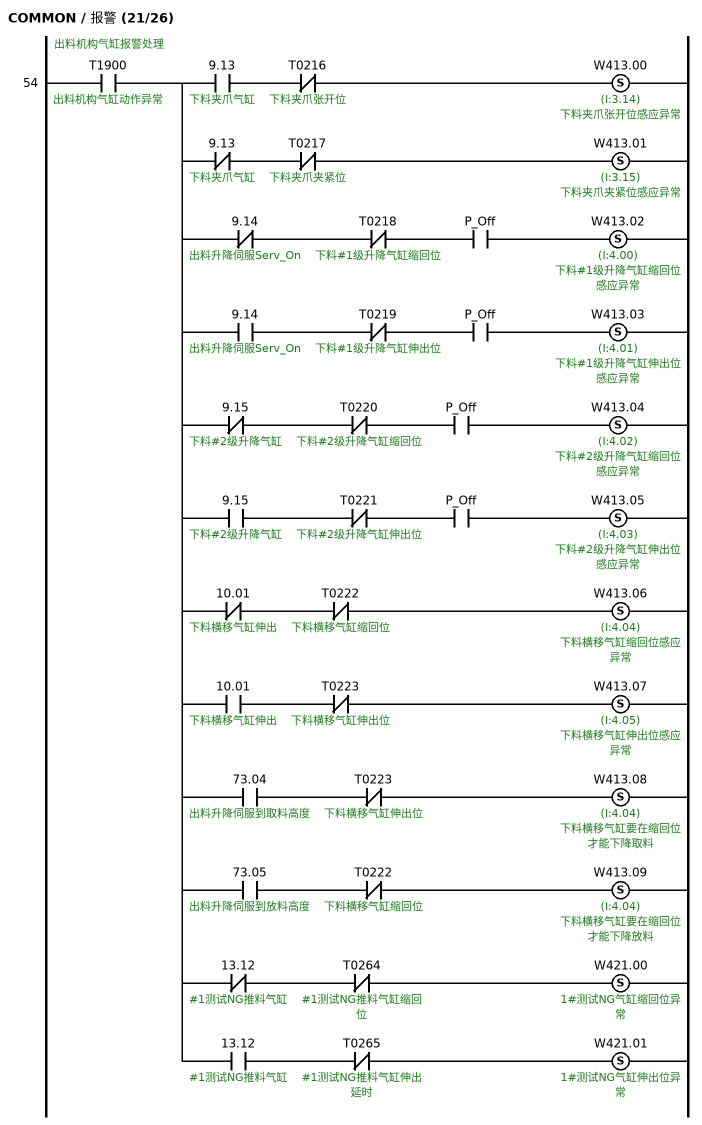
; [picture p456: COMMON / 报警, rungs 54-54]
; rung 54: 出料机构气缸报警处理
LD T1900  ; 出料机构气缸动作异常
OUT TR0
AND 9.13  ; 下料夹爪气缸
ANDNOT T0216  ; 下料夹爪张开位
SET W413.00  ; (I:3.14) 下料夹爪张开位感应异常
LD TR0
ANDNOT 9.13  ; 下料夹爪气缸
ANDNOT T0217  ; 下料夹爪夹紧位
SET W413.01  ; (I:3.15) 下料夹爪夹紧位感应异常
LD TR0
ANDNOT 9.14  ; 出料升降伺服Serv_On
ANDNOT T0218  ; 下料#1级升降气缸缩回位
AND P_Off
SET W413.02  ; (I:4.00) 下料#1级升降气缸缩回位感应异常
LD TR0
AND 9.14  ; 出料升降伺服Serv_On
ANDNOT T0219  ; 下料#1级升降气缸伸出位
AND P_Off
SET W413.03  ; (I:4.01) 下料#1级升降气缸伸出位感应异常
LD TR0
ANDNOT 9.15  ; 下料#2级升降气缸
ANDNOT T0220  ; 下料#2级升降气缸缩回位
AND P_Off
SET W413.04  ; (I:4.02) 下料#2级升降气缸缩回位感应异常
LD TR0
AND 9.15  ; 下料#2级升降气缸
ANDNOT T0221  ; 下料#2级升降气缸伸出位
AND P_Off
SET W413.05  ; (I:4.03) 下料#2级升降气缸伸出位感应异常
LD TR0
ANDNOT 10.01  ; 下料横移气缸伸出
ANDNOT T0222  ; 下料横移气缸缩回位
SET W413.06  ; (I:4.04) 下料横移气缸缩回位感应异常
LD TR0
AND 10.01  ; 下料横移气缸伸出
ANDNOT T0223  ; 下料横移气缸伸出位
SET W413.07  ; (I:4.05) 下料横移气缸伸出位感应异常
LD TR0
AND 73.04  ; 出料升降伺服到取料高度
ANDNOT T0223  ; 下料横移气缸伸出位
SET W413.08  ; (I:4.04) 下料横移气缸要在缩回位才能下降取料
LD TR0
AND 73.05  ; 出料升降伺服到放料高度
ANDNOT T0222  ; 下料横移气缸缩回位
SET W413.09  ; (I:4.04) 下料横移气缸要在缩回位才能下降放料
LD TR0
ANDNOT 13.12  ; #1测试NG推料气缸
ANDNOT T0264  ; #1测试NG推料气缸缩回位
SET W421.00  ; 1#测试NG气缸缩回位异常
LD TR0
AND 13.12  ; #1测试NG推料气缸
ANDNOT T0265  ; #1测试NG推料气缸伸出延时
SET W421.01  ; 1#测试NG气缸伸出位异常

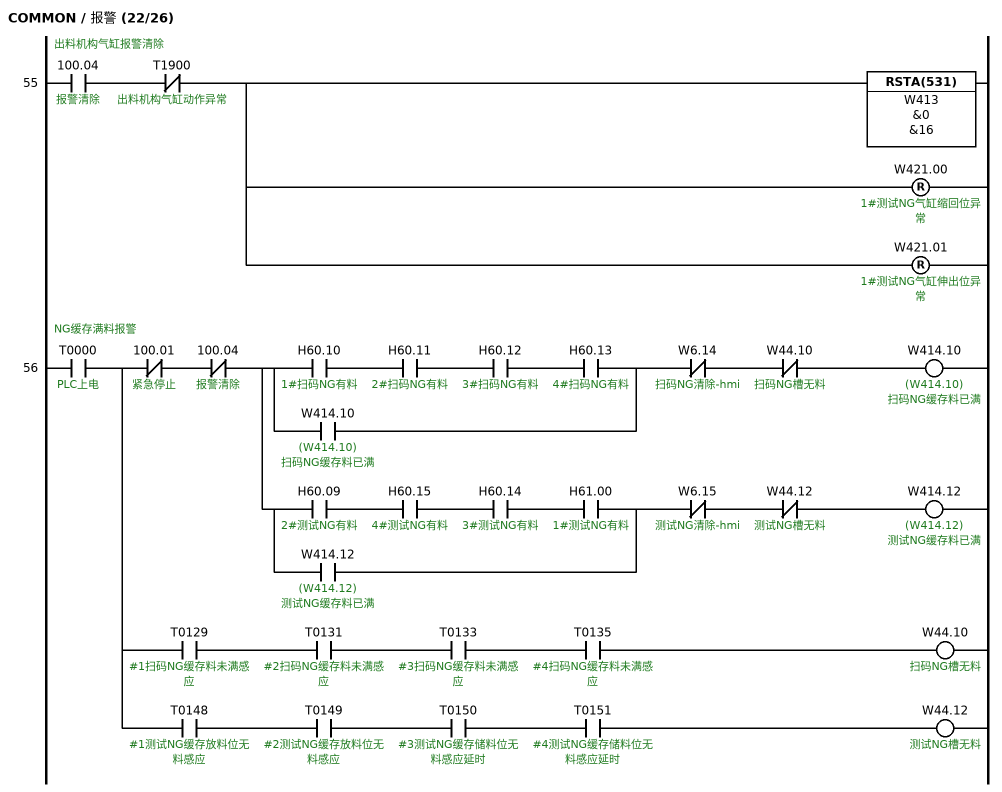
; rung 55: 出料机构气缸报警清除
LD 100.04  ; 报警清除
ANDNOT T1900  ; 出料机构气缸动作异常
RSTA(531) W413 &0 &16
RSET W421.00  ; 1#测试NG气缸缩回位异常
RSET W421.01  ; 1#测试NG气缸伸出位异常
; rung 56: NG缓存满料报警
LD T0000  ; PLC上电
OUT TR0
ANDNOT 100.01  ; 紧急停止
ANDNOT 100.04  ; 报警清除
OUT TR1
LD H60.10  ; 1#扫码NG有料
AND H60.11  ; 2#扫码NG有料
AND H60.12  ; 3#扫码NG有料
AND H60.13  ; 4#扫码NG有料
OR W414.10  ; (W414.10) 扫码NG缓存料已满
ANDLD
ANDNOT W6.14  ; 扫码NG清除-hmi
ANDNOT W44.10  ; 扫码NG槽无料
OUT W414.10  ; (W414.10) 扫码NG缓存料已满
LD TR1
LD H60.09  ; 2#测试NG有料
AND H60.15  ; 4#测试NG有料
AND H60.14  ; 3#测试NG有料
AND H61.00  ; 1#测试NG有料
OR W414.12  ; (W414.12) 测试NG缓存料已满
ANDLD
ANDNOT W6.15  ; 测试NG清除-hmi
ANDNOT W44.12  ; 测试NG槽无料
OUT W414.12  ; (W414.12) 测试NG缓存料已满
LD TR0
AND T0129  ; #1扫码NG缓存料未满感应
AND T0131  ; #2扫码NG缓存料未满感应
AND T0133  ; #3扫码NG缓存料未满感应
AND T0135  ; #4扫码NG缓存料未满感应
OUT W44.10  ; 扫码NG槽无料
LD TR0
AND T0148  ; #1测试NG缓存放料位无料感应
AND T0149  ; #2测试NG缓存放料位无料感应
AND T0150  ; #3测试NG缓存储料位无料感应延时
AND T0151  ; #4测试NG缓存储料位无料感应延时
OUT W44.12  ; 测试NG槽无料

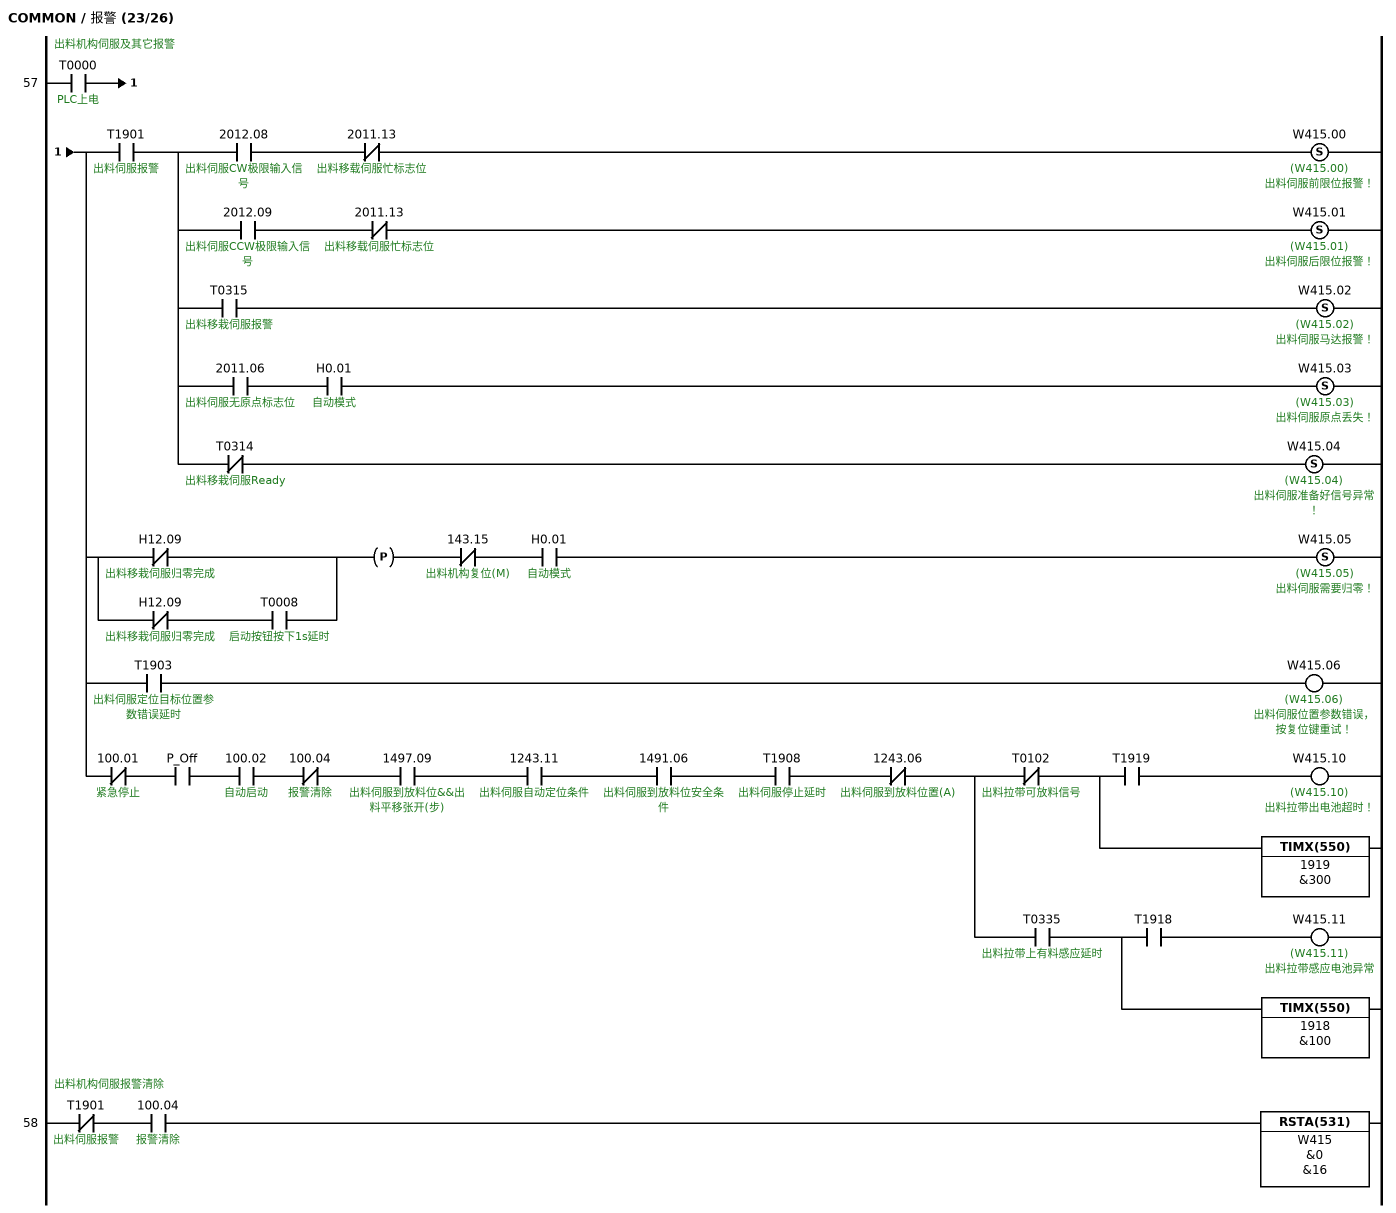
; rung 57: 出料机构伺服及其它报警
LD T0000  ; PLC上电
OUT TR0
AND T1901  ; 出料伺服报警
OUT TR1
AND 2012.08  ; 出料伺服CW极限输入信号
ANDNOT 2011.13  ; 出料移载伺服忙标志位
SET W415.00  ; (W415.00) 出料伺服前限位报警！
LD TR1
AND 2012.09  ; 出料伺服CCW极限输入信号
ANDNOT 2011.13  ; 出料移载伺服忙标志位
SET W415.01  ; (W415.01) 出料伺服后限位报警！
LD TR1
AND T0315  ; 出料移栽伺服报警
SET W415.02  ; (W415.02) 出料伺服马达报警！
LD TR1
AND 2011.06  ; 出料伺服无原点标志位
AND H0.01  ; 自动模式
SET W415.03  ; (W415.03) 出料伺服原点丢失！
LD TR1
ANDNOT T0314  ; 出料移栽伺服Ready
SET W415.04  ; (W415.04) 出料伺服准备好信号异常！
LD TR0
LDNOT H12.09  ; 出料移栽伺服归零完成
LDNOT H12.09  ; 出料移栽伺服归零完成
AND T0008  ; 启动按钮按下1s延时
ORLD
ANDLD
UP(521)
ANDNOT 143.15  ; 出料机构复位(M)
AND H0.01  ; 自动模式
SET W415.05  ; (W415.05) 出料伺服需要归零！
LD TR0
AND T1903  ; 出料伺服定位目标位置参数错误延时
OUT W415.06  ; (W415.06) 出料伺服位置参数错误，按复位键重试！
LD TR0
ANDNOT 100.01  ; 紧急停止
AND P_Off
AND 100.02  ; 自动启动
ANDNOT 100.04  ; 报警清除
AND 1497.09  ; 出料伺服到放料位&&出料平移张开(步)
AND 1243.11  ; 出料伺服自动定位条件
AND 1491.06  ; 出料伺服到放料位安全条件
AND T1908  ; 出料伺服停止延时
ANDNOT 1243.06  ; 出料伺服到放料位置(A)
OUT TR0
ANDNOT T0102  ; 出料拉带可放料信号
OUT TR1
AND T1919
OUT W415.10  ; (W415.10) 出料拉带出电池超时！
LD TR1
TIMX(550) 1919 &300
LD TR0
AND T0335  ; 出料拉带上有料感应延时
OUT TR0
AND T1918
OUT W415.11  ; (W415.11) 出料拉带感应电池异常
LD TR0
TIMX(550) 1918 &100
; rung 58: 出料机构伺服报警清除
LDNOT T1901  ; 出料伺服报警
AND 100.04  ; 报警清除
RSTA(531) W415 &0 &16

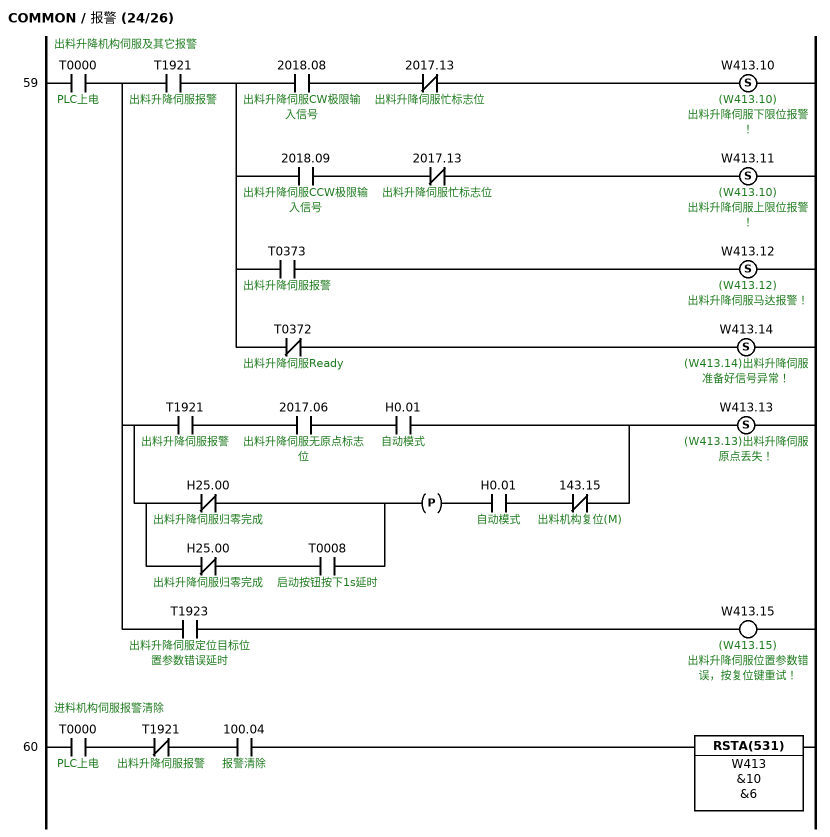
; rung 59: 出料升降机构伺服及其它报警
LD T0000  ; PLC上电
OUT TR0
AND T1921  ; 出料升降伺服报警
OUT TR1
AND 2018.08  ; 出料升降伺服CW极限输入信号
ANDNOT 2017.13  ; 出料升降伺服忙标志位
SET W413.10  ; (W413.10) 出料升降伺服下限位报警！
LD TR1
AND 2018.09  ; 出料升降伺服CCW极限输入信号
ANDNOT 2017.13  ; 出料升降伺服忙标志位
SET W413.11  ; (W413.10) 出料升降伺服上限位报警！
LD TR1
AND T0373  ; 出料升降伺服报警
SET W413.12  ; (W413.12) 出料升降伺服马达报警！
LD TR1
ANDNOT T0372  ; 出料升降伺服Ready
SET W413.14  ; (W413.14)出料升降伺服准备好信号异常！
LD TR0
LD T1921  ; 出料升降伺服报警
AND 2017.06  ; 出料升降伺服无原点标志位
AND H0.01  ; 自动模式
LDNOT H25.00  ; 出料升降伺服归零完成
LDNOT H25.00  ; 出料升降伺服归零完成
AND T0008  ; 启动按钮按下1s延时
ORLD
UP(521)
AND H0.01  ; 自动模式
ANDNOT 143.15  ; 出料机构复位(M)
ORLD
ANDLD
SET W413.13  ; (W413.13)出料升降伺服原点丢失！
LD TR0
AND T1923  ; 出料升降伺服定位目标位置参数错误延时
OUT W413.15  ; (W413.15) 出料升降伺服位置参数错误，按复位键重试！
; rung 60: 进料机构伺服报警清除
LD T0000  ; PLC上电
ANDNOT T1921  ; 出料升降伺服报警
AND 100.04  ; 报警清除
RSTA(531) W413 &10 &6

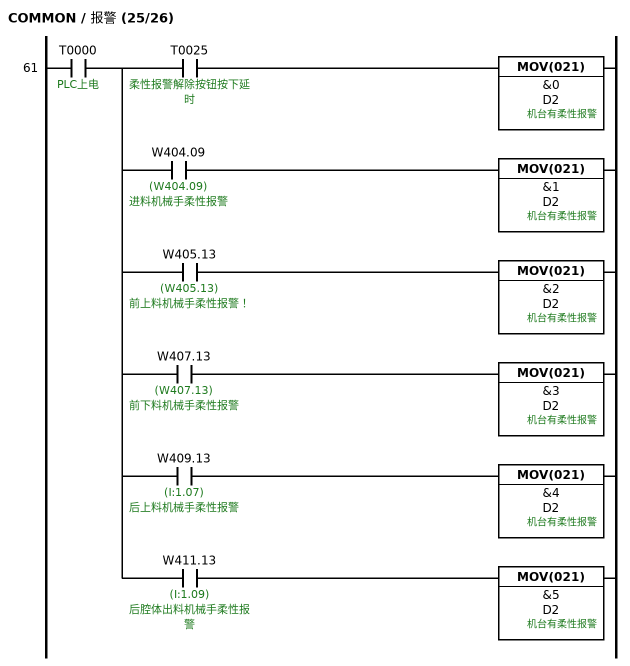
; rung 61
LD T0000  ; PLC上电
OUT TR0
AND T0025  ; 柔性报警解除按钮按下延时
MOV(021) &0 D2  ; 机台有柔性报警
LD TR0
AND W404.09  ; (W404.09) 进料机械手柔性报警
MOV(021) &1 D2  ; 机台有柔性报警
LD TR0
AND W405.13  ; (W405.13) 前上料机械手柔性报警！
MOV(021) &2 D2  ; 机台有柔性报警
LD TR0
AND W407.13  ; (W407.13) 前下料机械手柔性报警
MOV(021) &3 D2  ; 机台有柔性报警
LD TR0
AND W409.13  ; (I:1.07) 后上料机械手柔性报警
MOV(021) &4 D2  ; 机台有柔性报警
LD TR0
AND W411.13  ; (I:1.09) 后腔体出料机械手柔性报警
MOV(021) &5 D2  ; 机台有柔性报警

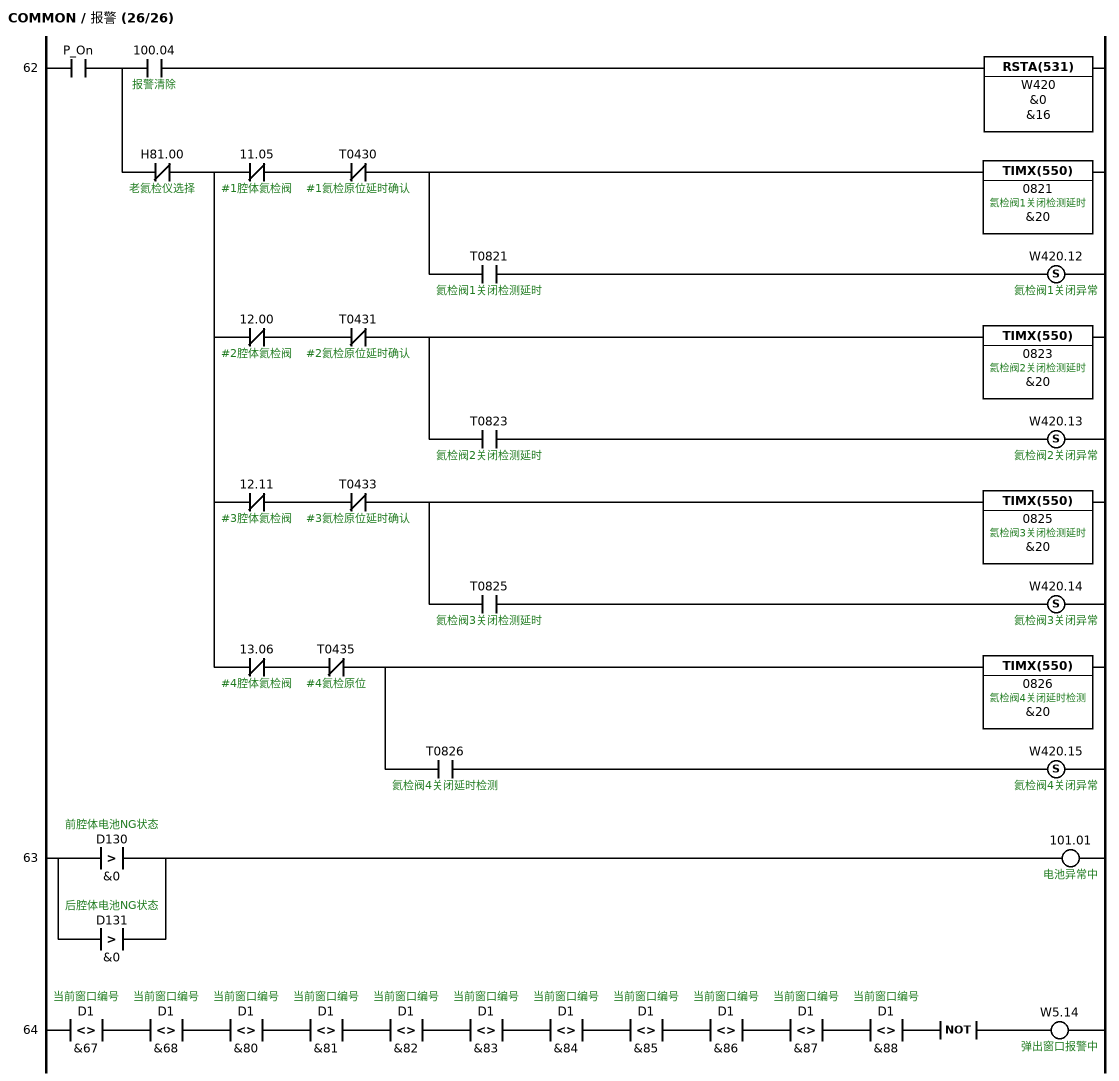
; rung 62
LD P_On
OUT TR0
AND 100.04  ; 报警清除
RSTA(531) W420 &0 &16
LD TR0
ANDNOT H81.00  ; 老氦检仪选择
OUT TR0
ANDNOT 11.05  ; #1腔体氦检阀
ANDNOT T0430  ; #1氦检原位延时确认
TIMX(550) 0821 &20  ; 氦检阀1关闭检测延时
AND T0821  ; 氦检阀1关闭检测延时
SET W420.12  ; 氦检阀1关闭异常
LD TR0
ANDNOT 12.00  ; #2腔体氦检阀
ANDNOT T0431  ; #2氦检原位延时确认
TIMX(550) 0823 &20  ; 氦检阀2关闭检测延时
AND T0823  ; 氦检阀2关闭检测延时
SET W420.13  ; 氦检阀2关闭异常
LD TR0
ANDNOT 12.11  ; #3腔体氦检阀
ANDNOT T0433  ; #3氦检原位延时确认
TIMX(550) 0825 &20  ; 氦检阀3关闭检测延时
AND T0825  ; 氦检阀3关闭检测延时
SET W420.14  ; 氦检阀3关闭异常
LD TR0
ANDNOT 13.06  ; #4腔体氦检阀
ANDNOT T0435  ; #4氦检原位
TIMX(550) 0826 &20  ; 氦检阀4关闭延时检测
AND T0826  ; 氦检阀4关闭延时检测
SET W420.15  ; 氦检阀4关闭异常
; rung 63
LD>(320) D130 &0  ; 前腔体电池NG状态
OR>(320) D131 &0  ; 后腔体电池NG状态
OUT 101.01  ; 电池异常中
; rung 64
LD<>(305) D1 &67  ; 当前窗口编号
AND<>(305) D1 &68  ; 当前窗口编号
AND<>(305) D1 &80  ; 当前窗口编号
AND<>(305) D1 &81  ; 当前窗口编号
AND<>(305) D1 &82  ; 当前窗口编号
AND<>(305) D1 &83  ; 当前窗口编号
AND<>(305) D1 &84  ; 当前窗口编号
AND<>(305) D1 &85  ; 当前窗口编号
AND<>(305) D1 &86  ; 当前窗口编号
AND<>(305) D1 &87  ; 当前窗口编号
AND<>(305) D1 &88  ; 当前窗口编号
NOT(520)
OUT W5.14  ; 弹出窗口报警中

### Section 数据传递

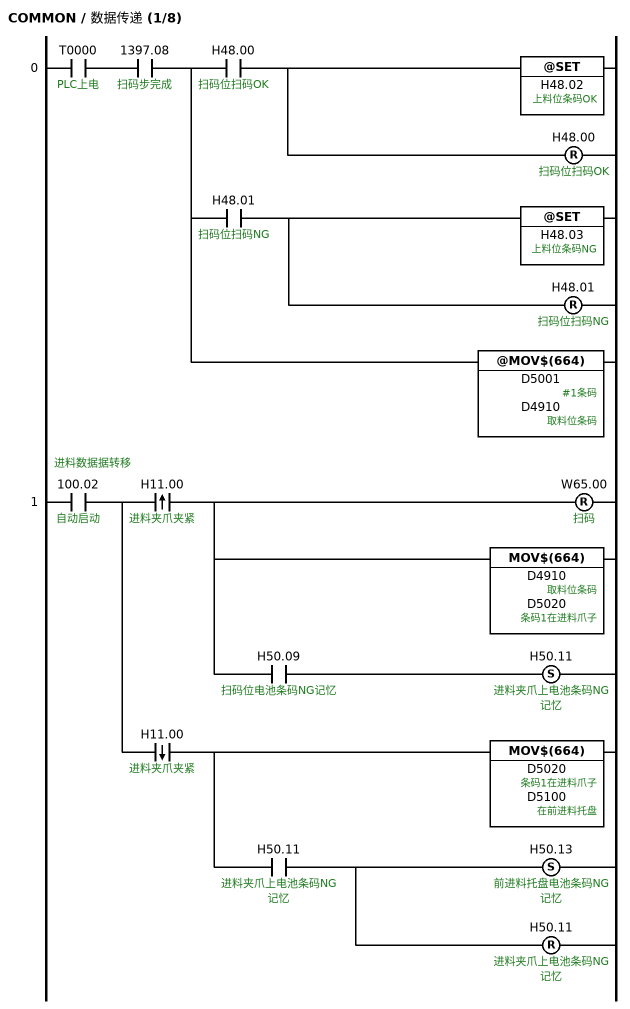
; rung 0
LD T0000  ; PLC上电
AND 1397.08  ; 扫码步完成
OUT TR0
AND H48.00  ; 扫码位扫码OK
@SET H48.02  ; 上料位条码OK
RSET H48.00  ; 扫码位扫码OK
LD TR0
AND H48.01  ; 扫码位扫码NG
@SET H48.03  ; 上料位条码NG
RSET H48.01  ; 扫码位扫码NG
LD TR0
@MOV$(664) D5001 D4910  ; #1条码, 取料位条码
; rung 1: 进料数据据转移
LD 100.02  ; 自动启动
OUT TR0
@AND H11.00  ; 进料夹爪夹紧
RSET W65.00  ; 扫码
MOV$(664) D4910 D5020  ; 取料位条码, 条码1在进料爪子
AND H50.09  ; 扫码位电池条码NG记忆
SET H50.11  ; 进料夹爪上电池条码NG记忆
LD TR0
%AND H11.00  ; 进料夹爪夹紧
MOV$(664) D5020 D5100  ; 条码1在进料爪子, 在前进料托盘
AND H50.11  ; 进料夹爪上电池条码NG记忆
SET H50.13  ; 前进料托盘电池条码NG记忆
RSET H50.11  ; 进料夹爪上电池条码NG记忆

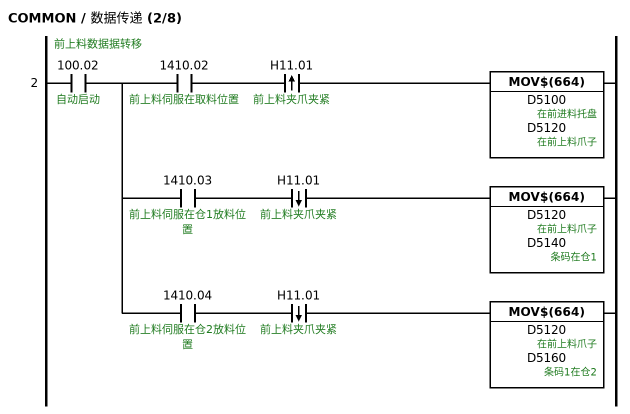
; rung 2: 前上料数据据转移
LD 100.02  ; 自动启动
OUT TR0
AND 1410.02  ; 前上料伺服在取料位置
@AND H11.01  ; 前上料夹爪夹紧
MOV$(664) D5100 D5120  ; 在前进料托盘, 在前上料爪子
LD TR0
AND 1410.03  ; 前上料伺服在仓1放料位置
%AND H11.01  ; 前上料夹爪夹紧
MOV$(664) D5120 D5140  ; 在前上料爪子, 条码在仓1
LD TR0
AND 1410.04  ; 前上料伺服在仓2放料位置
%AND H11.01  ; 前上料夹爪夹紧
MOV$(664) D5120 D5160  ; 在前上料爪子, 条码1在仓2

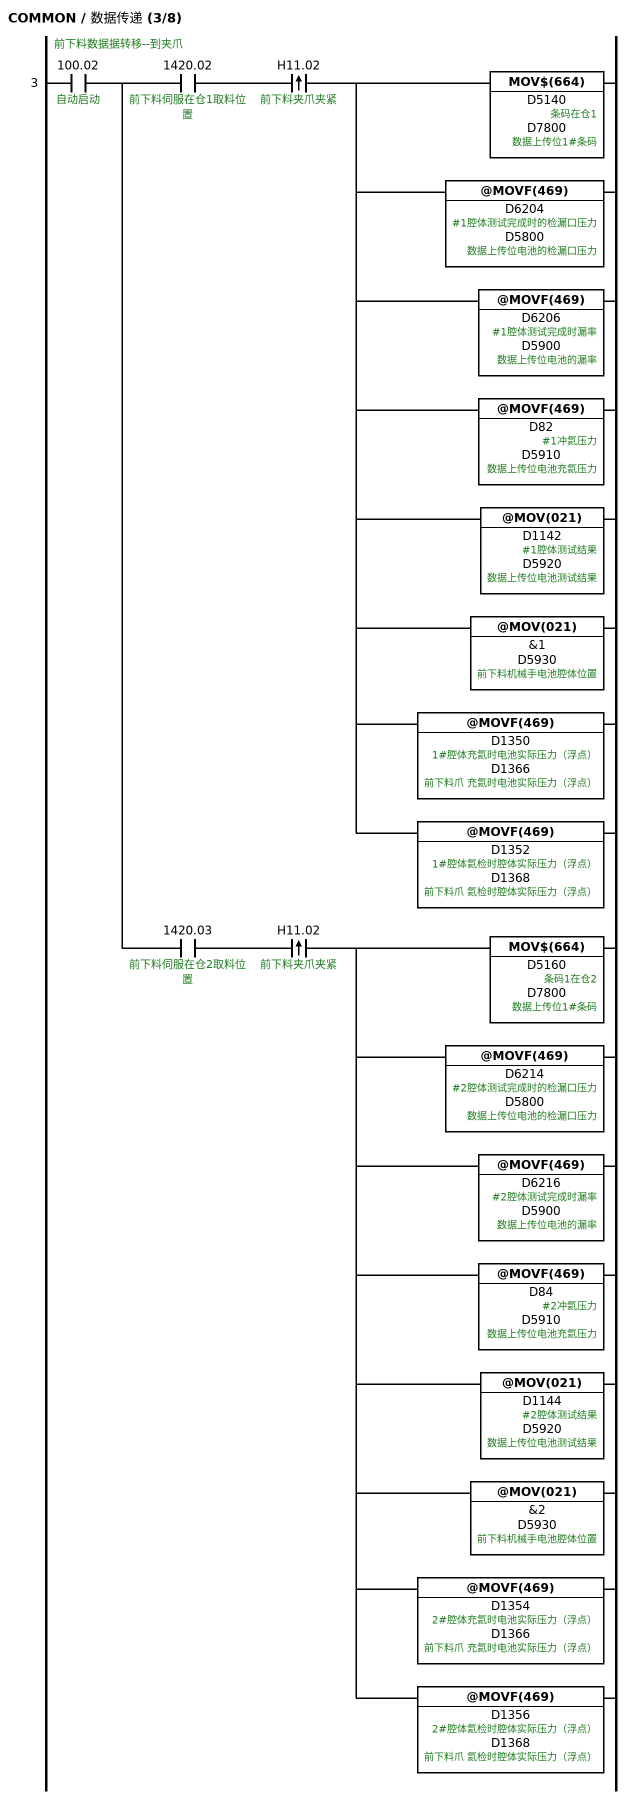
; rung 3: 前下料数据据转移--到夹爪
LD 100.02  ; 自动启动
OUT TR0
AND 1420.02  ; 前下料伺服在仓1取料位置
@AND H11.02  ; 前下料夹爪夹紧
MOV$(664) D5140 D7800  ; 条码在仓1, 数据上传位1#条码
@MOVF(469) D6204 D5800  ; #1腔体测试完成时的检漏口压力, 数据上传位电池的检漏口压力
@MOVF(469) D6206 D5900  ; #1腔体测试完成时漏率, 数据上传位电池的漏率
@MOVF(469) D82 D5910  ; #1冲氦压力, 数据上传位电池充氦压力
@MOV(021) D1142 D5920  ; #1腔体测试结果, 数据上传位电池测试结果
@MOV(021) &1 D5930  ; 前下料机械手电池腔体位置
@MOVF(469) D1350 D1366  ; 1#腔体充氦时电池实际压力（浮点）, 前下料爪 充氦时电池实际压力（浮点）
@MOVF(469) D1352 D1368  ; 1#腔体氦检时腔体实际压力（浮点）, 前下料爪 氦检时腔体实际压力（浮点）
LD TR0
AND 1420.03  ; 前下料伺服在仓2取料位置
@AND H11.02  ; 前下料夹爪夹紧
MOV$(664) D5160 D7800  ; 条码1在仓2, 数据上传位1#条码
@MOVF(469) D6214 D5800  ; #2腔体测试完成时的检漏口压力, 数据上传位电池的检漏口压力
@MOVF(469) D6216 D5900  ; #2腔体测试完成时漏率, 数据上传位电池的漏率
@MOVF(469) D84 D5910  ; #2冲氦压力, 数据上传位电池充氦压力
@MOV(021) D1144 D5920  ; #2腔体测试结果, 数据上传位电池测试结果
@MOV(021) &2 D5930  ; 前下料机械手电池腔体位置
@MOVF(469) D1354 D1366  ; 2#腔体充氦时电池实际压力（浮点）, 前下料爪 充氦时电池实际压力（浮点）
@MOVF(469) D1356 D1368  ; 2#腔体氦检时腔体实际压力（浮点）, 前下料爪 氦检时腔体实际压力（浮点）

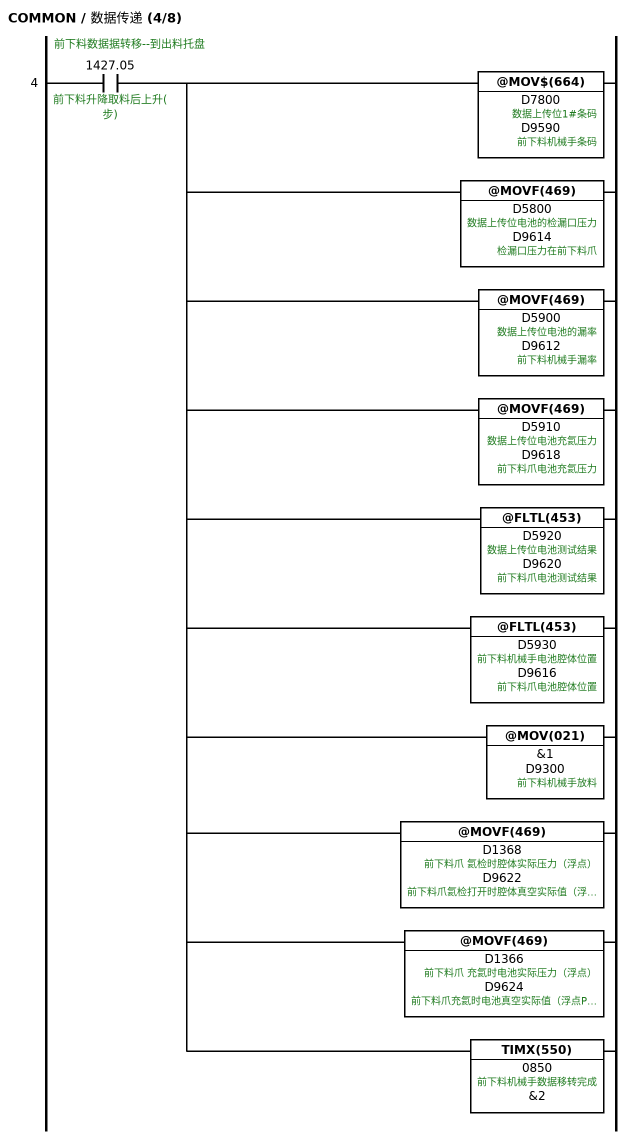
; rung 4: 前下料数据据转移--到出料托盘
LD 1427.05  ; 前下料升降取料后上升(步)
@MOV$(664) D7800 D9590  ; 数据上传位1#条码, 前下料机械手条码
@MOVF(469) D5800 D9614  ; 数据上传位电池的检漏口压力, 检漏口压力在前下料爪
@MOVF(469) D5900 D9612  ; 数据上传位电池的漏率, 前下料机械手漏率
@MOVF(469) D5910 D9618  ; 数据上传位电池充氦压力, 前下料爪电池充氦压力
@FLTL(453) D5920 D9620  ; 数据上传位电池测试结果, 前下料爪电池测试结果
@FLTL(453) D5930 D9616  ; 前下料机械手电池腔体位置, 前下料爪电池腔体位置
@MOV(021) &1 D9300  ; 前下料机械手放料
@MOVF(469) D1368 D9622  ; 前下料爪 氦检时腔体实际压力（浮点）, 前下料爪氦检打开时腔体真空实际值（浮点PC）
@MOVF(469) D1366 D9624  ; 前下料爪 充氦时电池实际压力（浮点）, 前下料爪充氦时电池真空实际值（浮点PC）
TIMX(550) 0850 &2  ; 前下料机械手数据移转完成

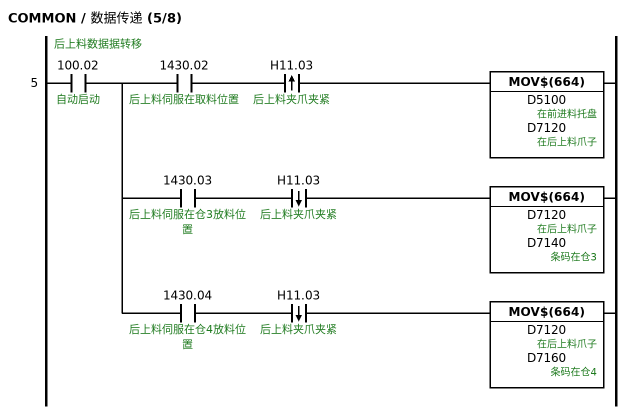
; rung 5: 后上料数据据转移
LD 100.02  ; 自动启动
OUT TR0
AND 1430.02  ; 后上料伺服在取料位置
@AND H11.03  ; 后上料夹爪夹紧
MOV$(664) D5100 D7120  ; 在前进料托盘, 在后上料爪子
LD TR0
AND 1430.03  ; 后上料伺服在仓3放料位置
%AND H11.03  ; 后上料夹爪夹紧
MOV$(664) D7120 D7140  ; 在后上料爪子, 条码在仓3
LD TR0
AND 1430.04  ; 后上料伺服在仓4放料位置
%AND H11.03  ; 后上料夹爪夹紧
MOV$(664) D7120 D7160  ; 在后上料爪子, 条码在仓4

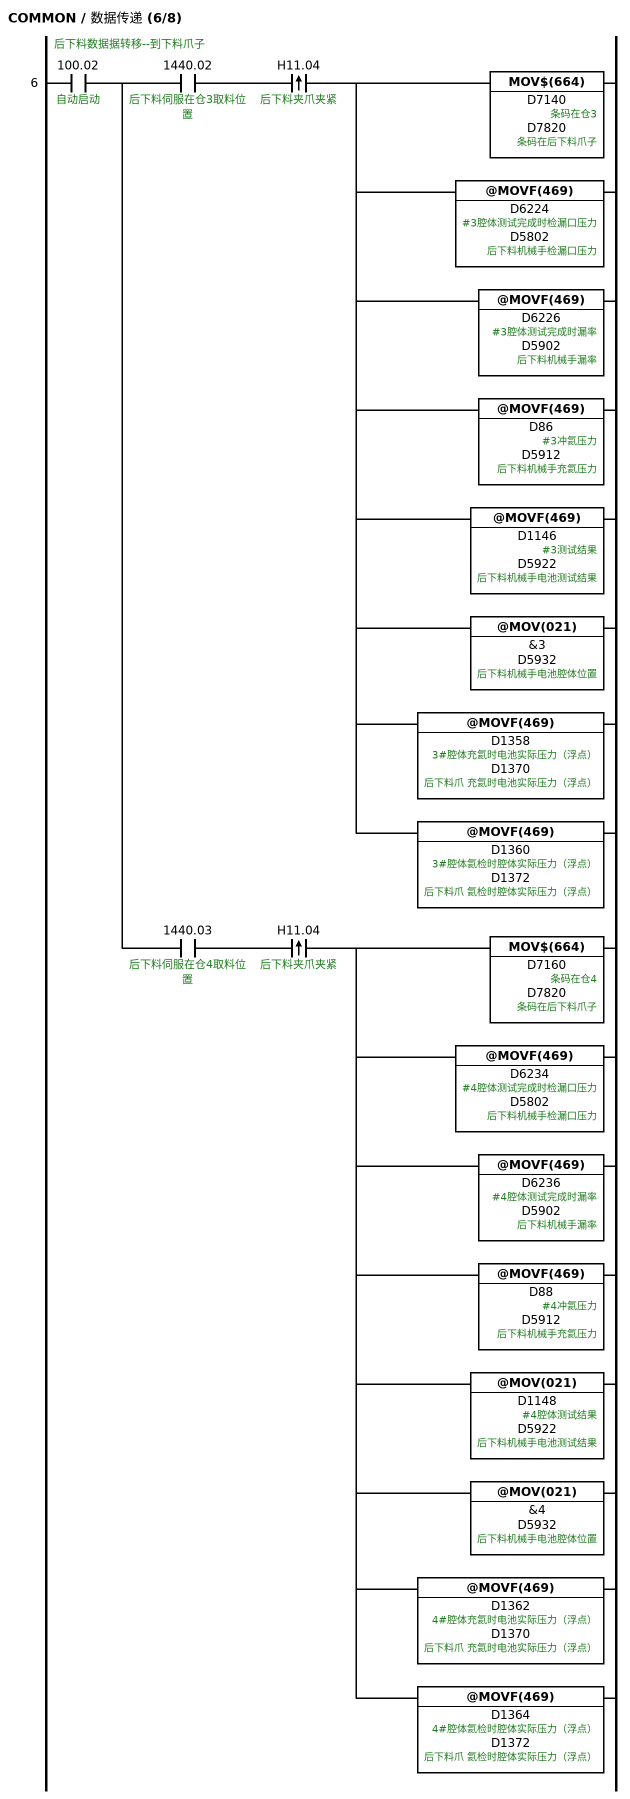
; rung 6: 后下料数据据转移--到下料爪子
LD 100.02  ; 自动启动
OUT TR0
AND 1440.02  ; 后下料伺服在仓3取料位置
@AND H11.04  ; 后下料夹爪夹紧
MOV$(664) D7140 D7820  ; 条码在仓3, 条码在后下料爪子
@MOVF(469) D6224 D5802  ; #3腔体测试完成时检漏口压力, 后下料机械手检漏口压力
@MOVF(469) D6226 D5902  ; #3腔体测试完成时漏率, 后下料机械手漏率
@MOVF(469) D86 D5912  ; #3冲氦压力, 后下料机械手充氦压力
@MOVF(469) D1146 D5922  ; #3测试结果, 后下料机械手电池测试结果
@MOV(021) &3 D5932  ; 后下料机械手电池腔体位置
@MOVF(469) D1358 D1370  ; 3#腔体充氦时电池实际压力（浮点）, 后下料爪 充氦时电池实际压力（浮点）
@MOVF(469) D1360 D1372  ; 3#腔体氦检时腔体实际压力（浮点）, 后下料爪 氦检时腔体实际压力（浮点）
LD TR0
AND 1440.03  ; 后下料伺服在仓4取料位置
@AND H11.04  ; 后下料夹爪夹紧
MOV$(664) D7160 D7820  ; 条码在仓4, 条码在后下料爪子
@MOVF(469) D6234 D5802  ; #4腔体测试完成时检漏口压力, 后下料机械手检漏口压力
@MOVF(469) D6236 D5902  ; #4腔体测试完成时漏率, 后下料机械手漏率
@MOVF(469) D88 D5912  ; #4冲氦压力, 后下料机械手充氦压力
@MOV(021) D1148 D5922  ; #4腔体测试结果, 后下料机械手电池测试结果
@MOV(021) &4 D5932  ; 后下料机械手电池腔体位置
@MOVF(469) D1362 D1370  ; 4#腔体充氦时电池实际压力（浮点）, 后下料爪 充氦时电池实际压力（浮点）
@MOVF(469) D1364 D1372  ; 4#腔体氦检时腔体实际压力（浮点）, 后下料爪 氦检时腔体实际压力（浮点）

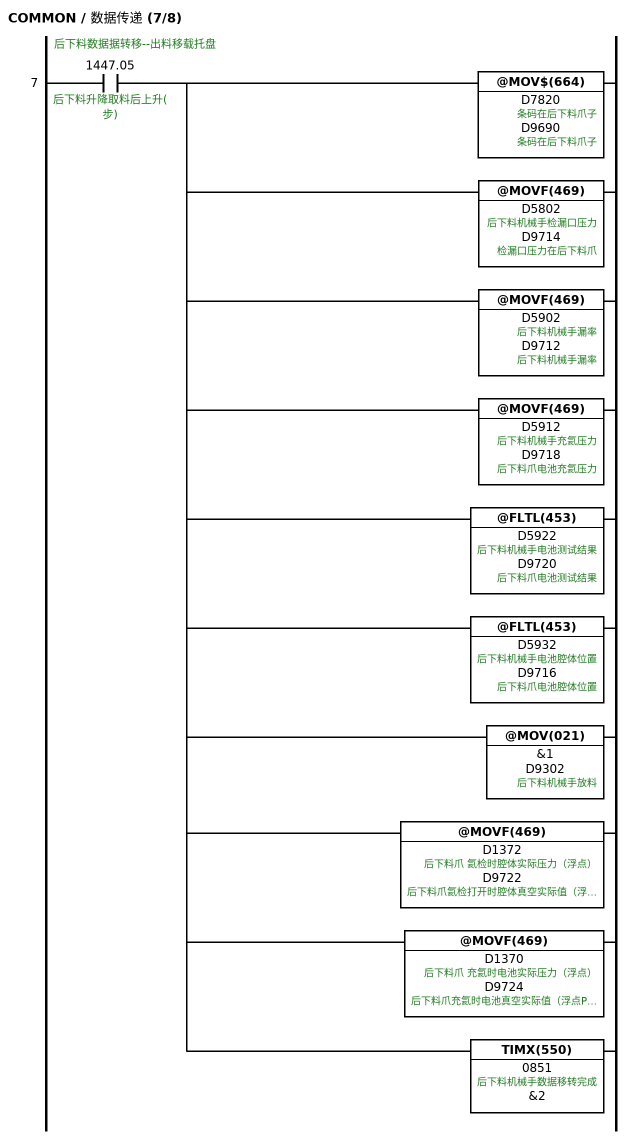
; rung 7: 后下料数据据转移--出料移载托盘
LD 1447.05  ; 后下料升降取料后上升(步)
@MOV$(664) D7820 D9690  ; 条码在后下料爪子
@MOVF(469) D5802 D9714  ; 后下料机械手检漏口压力, 检漏口压力在后下料爪
@MOVF(469) D5902 D9712  ; 后下料机械手漏率
@MOVF(469) D5912 D9718  ; 后下料机械手充氦压力, 后下料爪电池充氦压力
@FLTL(453) D5922 D9720  ; 后下料机械手电池测试结果, 后下料爪电池测试结果
@FLTL(453) D5932 D9716  ; 后下料机械手电池腔体位置, 后下料爪电池腔体位置
@MOV(021) &1 D9302  ; 后下料机械手放料
@MOVF(469) D1372 D9722  ; 后下料爪 氦检时腔体实际压力（浮点）, 后下料爪氦检打开时腔体真空实际值（浮点PC）
@MOVF(469) D1370 D9724  ; 后下料爪 充氦时电池实际压力（浮点）, 后下料爪充氦时电池真空实际值（浮点PC）
TIMX(550) 0851 &2  ; 后下料机械手数据移转完成

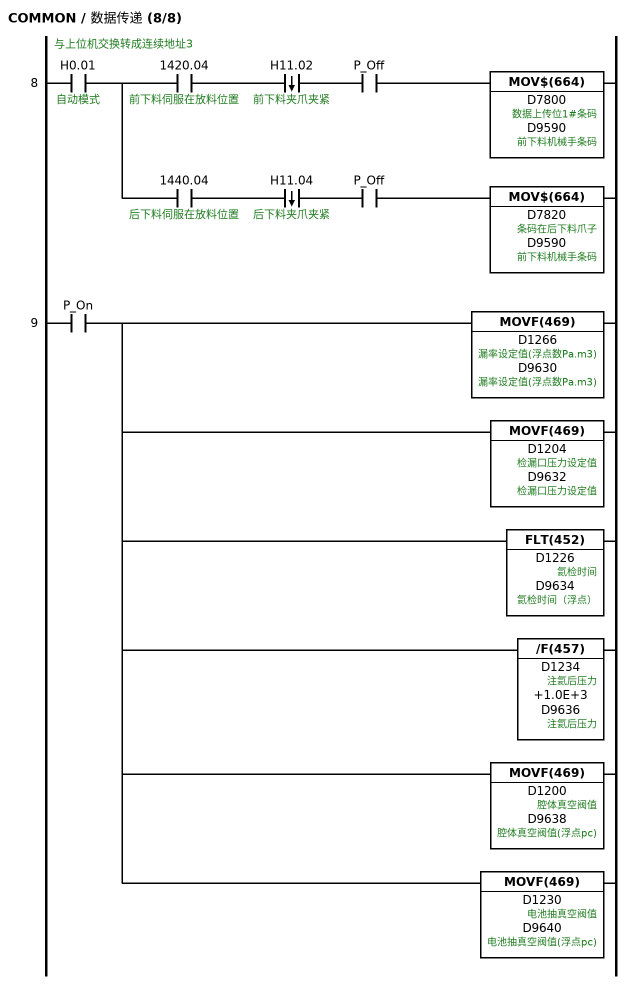
; rung 8: 与上位机交换转成连续地址3
LD H0.01  ; 自动模式
OUT TR0
AND 1420.04  ; 前下料伺服在放料位置
%AND H11.02  ; 前下料夹爪夹紧
AND P_Off
MOV$(664) D7800 D9590  ; 数据上传位1#条码, 前下料机械手条码
LD TR0
AND 1440.04  ; 后下料伺服在放料位置
%AND H11.04  ; 后下料夹爪夹紧
AND P_Off
MOV$(664) D7820 D9590  ; 条码在后下料爪子, 前下料机械手条码
; rung 9
LD P_On
MOVF(469) D1266 D9630  ; 漏率设定值(浮点数Pa.m3)
MOVF(469) D1204 D9632  ; 检漏口压力设定值
FLT(452) D1226 D9634  ; 氦检时间, 氦检时间（浮点）
/F(457) D1234 +1.0E+3 D9636  ; 注氦后压力
MOVF(469) D1200 D9638  ; 腔体真空阀值, 腔体真空阀值(浮点pc)
MOVF(469) D1230 D9640  ; 电池抽真空阀值, 电池抽真空阀值(浮点pc)

### Section PC交互

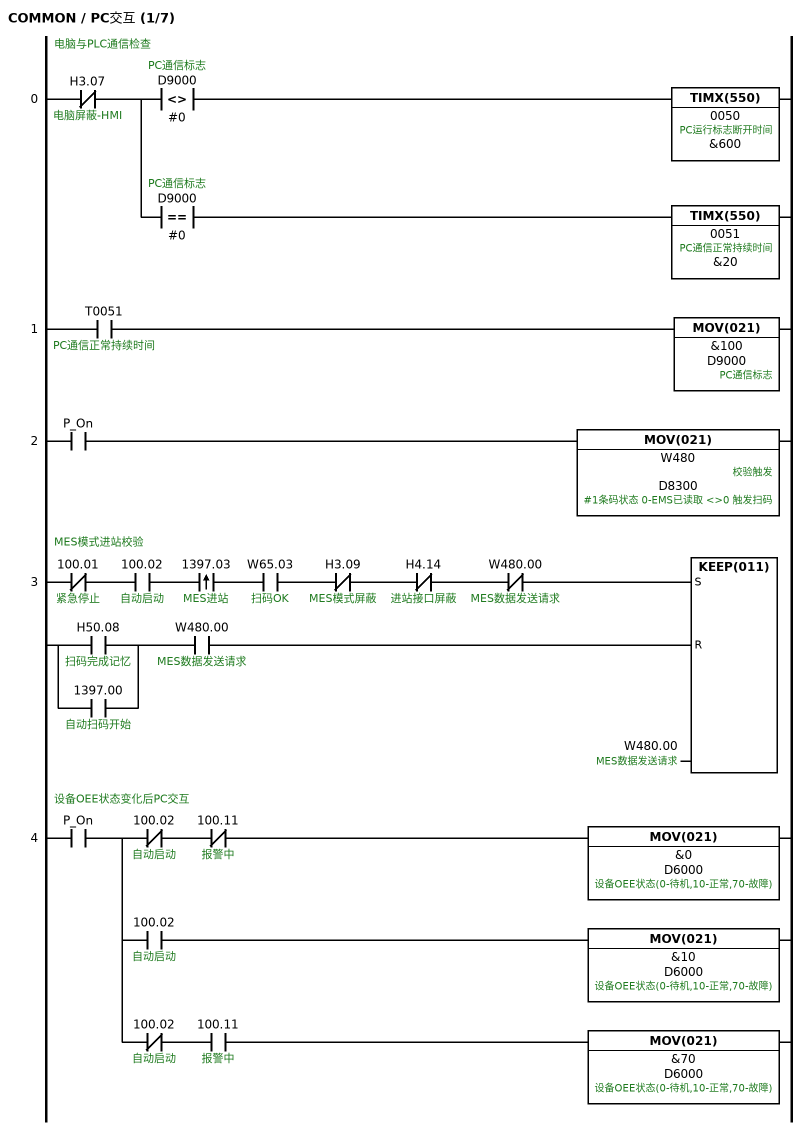
; rung 0: 电脑与PLC通信检查
LDNOT H3.07  ; 电脑屏蔽-HMI
OUT TR0
AND<>(305) D9000 #0  ; PC通信标志
TIMX(550) 0050 &600  ; PC运行标志断开时间
LD TR0
AND=(300) D9000 #0  ; PC通信标志
TIMX(550) 0051 &20  ; PC通信正常持续时间
; rung 1
LD T0051  ; PC通信正常持续时间
MOV(021) &100 D9000  ; PC通信标志
; rung 2
LD P_On
MOV(021) W480 D8300  ; 校验触发, #1条码状态 0-EMS已读取 <>0 触发扫码
; rung 3: MES模式进站校验
LDNOT 100.01  ; 紧急停止
AND 100.02  ; 自动启动
@AND 1397.03  ; MES进站
AND W65.03  ; 扫码OK
ANDNOT H3.09  ; MES模式屏蔽
ANDNOT H4.14  ; 进站接口屏蔽
ANDNOT W480.00  ; MES数据发送请求
LD H50.08  ; 扫码完成记忆
OR 1397.00  ; 自动扫码开始
AND W480.00  ; MES数据发送请求
KEEP(011) W480.00  ; MES数据发送请求
; rung 4: 设备OEE状态变化后PC交互
LD P_On
OUT TR0
ANDNOT 100.02  ; 自动启动
ANDNOT 100.11  ; 报警中
MOV(021) &0 D6000  ; 设备OEE状态(0-待机,10-正常,70-故障)
LD TR0
AND 100.02  ; 自动启动
MOV(021) &10 D6000  ; 设备OEE状态(0-待机,10-正常,70-故障)
LD TR0
ANDNOT 100.02  ; 自动启动
AND 100.11  ; 报警中
MOV(021) &70 D6000  ; 设备OEE状态(0-待机,10-正常,70-故障)

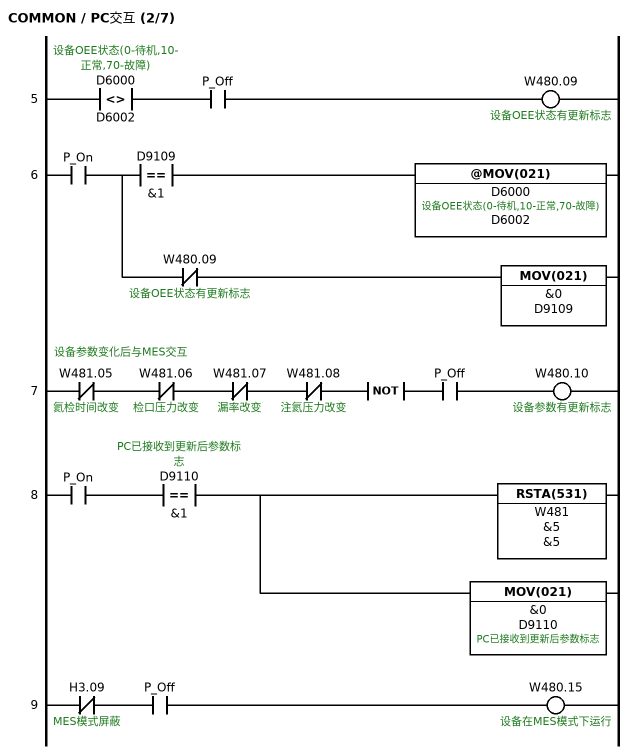
; rung 5
LD<>(305) D6000 D6002  ; 设备OEE状态(0-待机,10-正常,70-故障)
AND P_Off
OUT W480.09  ; 设备OEE状态有更新标志
; rung 6
LD P_On
OUT TR0
AND=(300) D9109 &1
@MOV(021) D6000 D6002  ; 设备OEE状态(0-待机,10-正常,70-故障)
LD TR0
ANDNOT W480.09  ; 设备OEE状态有更新标志
MOV(021) &0 D9109
; rung 7: 设备参数变化后与MES交互
LDNOT W481.05  ; 氦检时间改变
ANDNOT W481.06  ; 检口压力改变
ANDNOT W481.07  ; 漏率改变
ANDNOT W481.08  ; 注氦压力改变
NOT(520)
AND P_Off
OUT W480.10  ; 设备参数有更新标志
; rung 8
LD P_On
AND=(300) D9110 &1  ; PC已接收到更新后参数标志
RSTA(531) W481 &5 &5
MOV(021) &0 D9110  ; PC已接收到更新后参数标志
; rung 9
LDNOT H3.09  ; MES模式屏蔽
AND P_Off
OUT W480.15  ; 设备在MES模式下运行

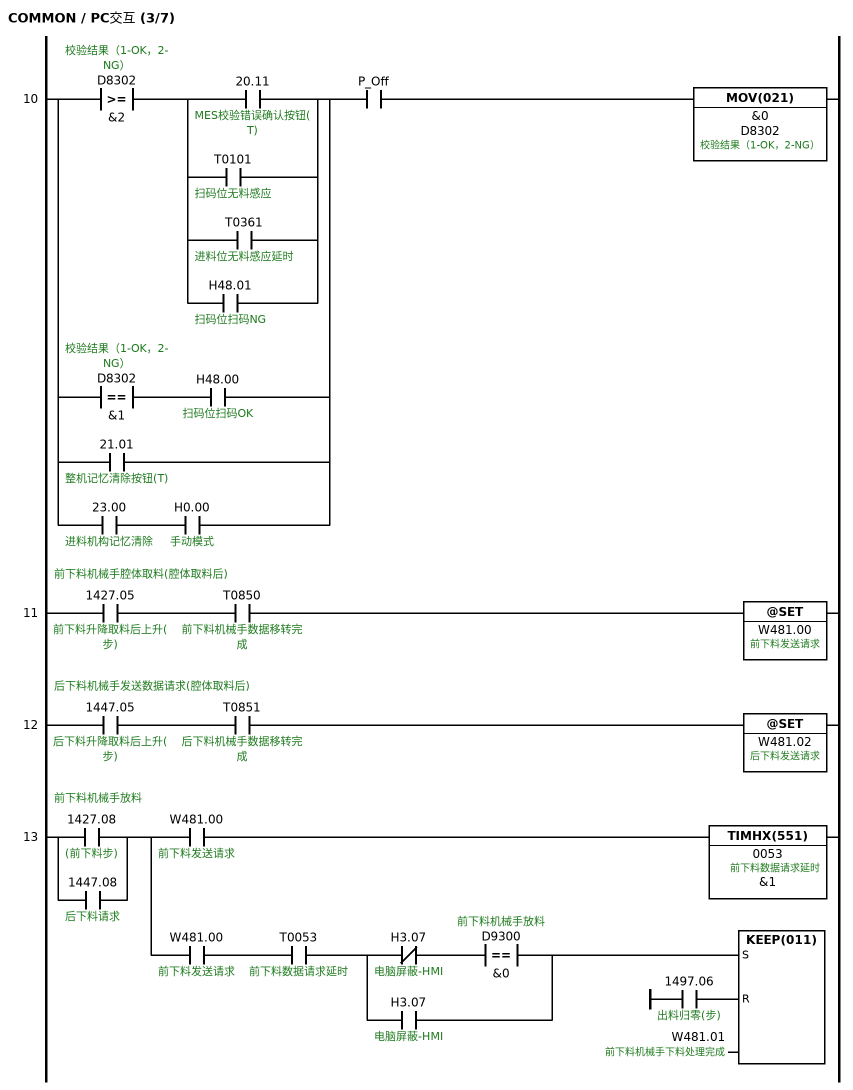
; rung 10
LD>=(325) D8302 &2  ; 校验结果（1-OK，2-NG）
LD 20.11  ; MES校验错误确认按钮(T)
OR T0101  ; 扫码位无料感应
OR T0361  ; 进料位无料感应延时
OR H48.01  ; 扫码位扫码NG
ANDLD
LD=(300) D8302 &1  ; 校验结果（1-OK，2-NG）
AND H48.00  ; 扫码位扫码OK
ORLD
OR 21.01  ; 整机记忆清除按钮(T)
LD 23.00  ; 进料机构记忆清除
AND H0.00  ; 手动模式
ORLD
AND P_Off
MOV(021) &0 D8302  ; 校验结果（1-OK，2-NG）
; rung 11: 前下料机械手腔体取料(腔体取料后)
LD 1427.05  ; 前下料升降取料后上升(步)
AND T0850  ; 前下料机械手数据移转完成
@SET W481.00  ; 前下料发送请求
; rung 12: 后下料机械手发送数据请求(腔体取料后)
LD 1447.05  ; 后下料升降取料后上升(步)
AND T0851  ; 后下料机械手数据移转完成
@SET W481.02  ; 后下料发送请求
; rung 13: 前下料机械手放料
LD 1427.08  ; (前下料步)
OR 1447.08  ; 后下料请求
OUT TR0
AND W481.00  ; 前下料发送请求
TIMHX(551) 0053 &1  ; 前下料数据请求延时
LD TR0
AND W481.00  ; 前下料发送请求
AND T0053  ; 前下料数据请求延时
LDNOT H3.07  ; 电脑屏蔽-HMI
AND=(300) D9300 &0  ; 前下料机械手放料
OR H3.07  ; 电脑屏蔽-HMI
ANDLD
LD 1497.06  ; 出料归零(步)
KEEP(011) W481.01  ; 前下料机械手下料处理完成

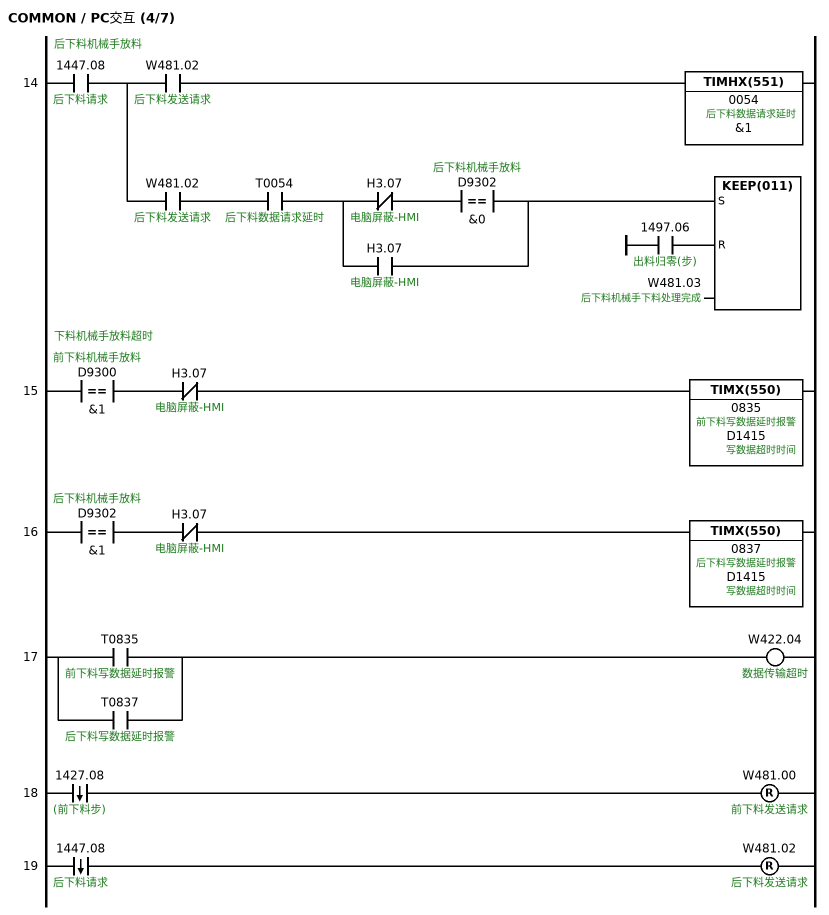
; rung 14: 后下料机械手放料
LD 1447.08  ; 后下料请求
OUT TR0
AND W481.02  ; 后下料发送请求
TIMHX(551) 0054 &1  ; 后下料数据请求延时
LD TR0
AND W481.02  ; 后下料发送请求
AND T0054  ; 后下料数据请求延时
LDNOT H3.07  ; 电脑屏蔽-HMI
AND=(300) D9302 &0  ; 后下料机械手放料
OR H3.07  ; 电脑屏蔽-HMI
ANDLD
LD 1497.06  ; 出料归零(步)
KEEP(011) W481.03  ; 后下料机械手下料处理完成
; rung 15: 下料机械手放料超时
LD=(300) D9300 &1  ; 前下料机械手放料
ANDNOT H3.07  ; 电脑屏蔽-HMI
TIMX(550) 0835 D1415  ; 写数据超时时间, 前下料写数据延时报警
; rung 16
LD=(300) D9302 &1  ; 后下料机械手放料
ANDNOT H3.07  ; 电脑屏蔽-HMI
TIMX(550) 0837 D1415  ; 写数据超时时间, 后下料写数据延时报警
; rung 17
LD T0835  ; 前下料写数据延时报警
OR T0837  ; 后下料写数据延时报警
OUT W422.04  ; 数据传输超时
; rung 18
%LD 1427.08  ; (前下料步)
RSET W481.00  ; 前下料发送请求
; rung 19
%LD 1447.08  ; 后下料请求
RSET W481.02  ; 后下料发送请求

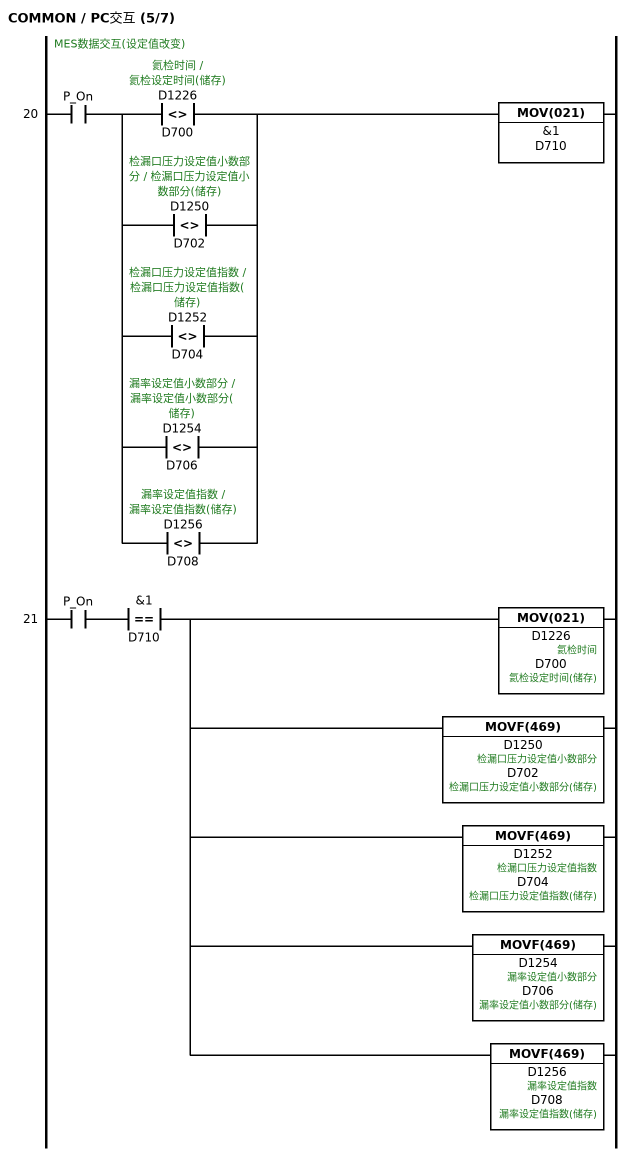
; rung 20: MES数据交互(设定值改变)
LD P_On
LD<>(305) D1226 D700  ; 氦检时间, 氦检设定时间(储存)
OR<>F(330) D1250 D702  ; 检漏口压力设定值小数部分, 检漏口压力设定值小数部分(储存)
OR<>F(330) D1252 D704  ; 检漏口压力设定值指数, 检漏口压力设定值指数(储存)
OR<>F(330) D1254 D706  ; 漏率设定值小数部分, 漏率设定值小数部分(储存)
OR<>F(330) D1256 D708  ; 漏率设定值指数, 漏率设定值指数(储存)
ANDLD
MOV(021) &1 D710
; rung 21
LD P_On
AND=(300) &1 D710
MOV(021) D1226 D700  ; 氦检时间, 氦检设定时间(储存)
MOVF(469) D1250 D702  ; 检漏口压力设定值小数部分, 检漏口压力设定值小数部分(储存)
MOVF(469) D1252 D704  ; 检漏口压力设定值指数, 检漏口压力设定值指数(储存)
MOVF(469) D1254 D706  ; 漏率设定值小数部分, 漏率设定值小数部分(储存)
MOVF(469) D1256 D708  ; 漏率设定值指数, 漏率设定值指数(储存)

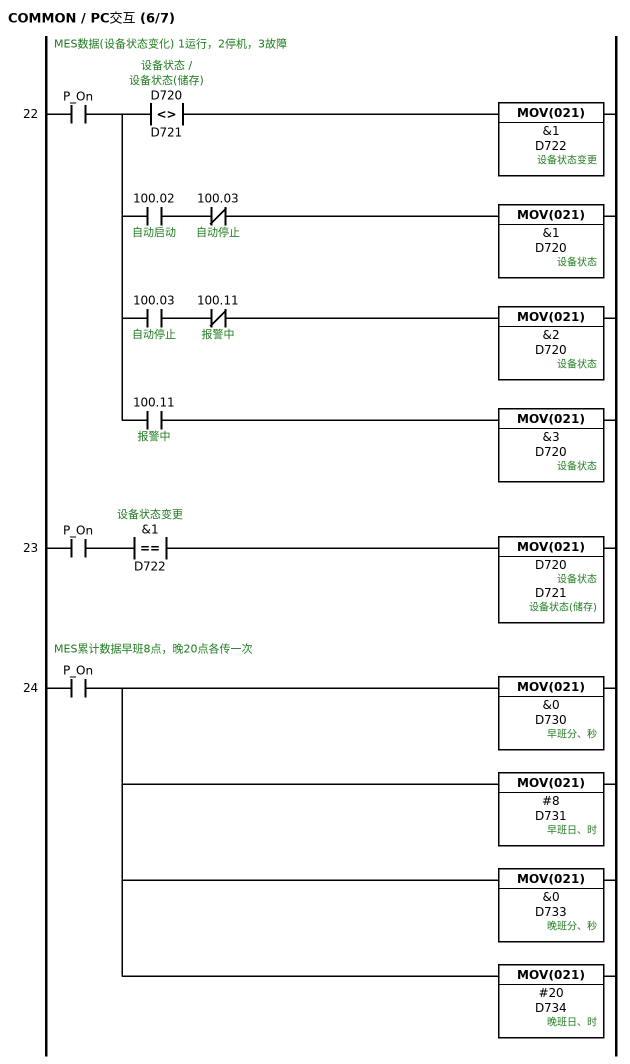
; rung 22: MES数据(设备状态变化) 1运行，2停机，3故障
LD P_On
OUT TR0
AND<>(305) D720 D721  ; 设备状态, 设备状态(储存)
MOV(021) &1 D722  ; 设备状态变更
LD TR0
AND 100.02  ; 自动启动
ANDNOT 100.03  ; 自动停止
MOV(021) &1 D720  ; 设备状态
LD TR0
AND 100.03  ; 自动停止
ANDNOT 100.11  ; 报警中
MOV(021) &2 D720  ; 设备状态
LD TR0
AND 100.11  ; 报警中
MOV(021) &3 D720  ; 设备状态
; rung 23
LD P_On
AND=(300) &1 D722  ; 设备状态变更
MOV(021) D720 D721  ; 设备状态, 设备状态(储存)
; rung 24: MES累计数据早班8点，晚20点各传一次
LD P_On
MOV(021) &0 D730  ; 早班分、秒
MOV(021) #8 D731  ; 早班日、时
MOV(021) &0 D733  ; 晚班分、秒
MOV(021) #20 D734  ; 晚班日、时

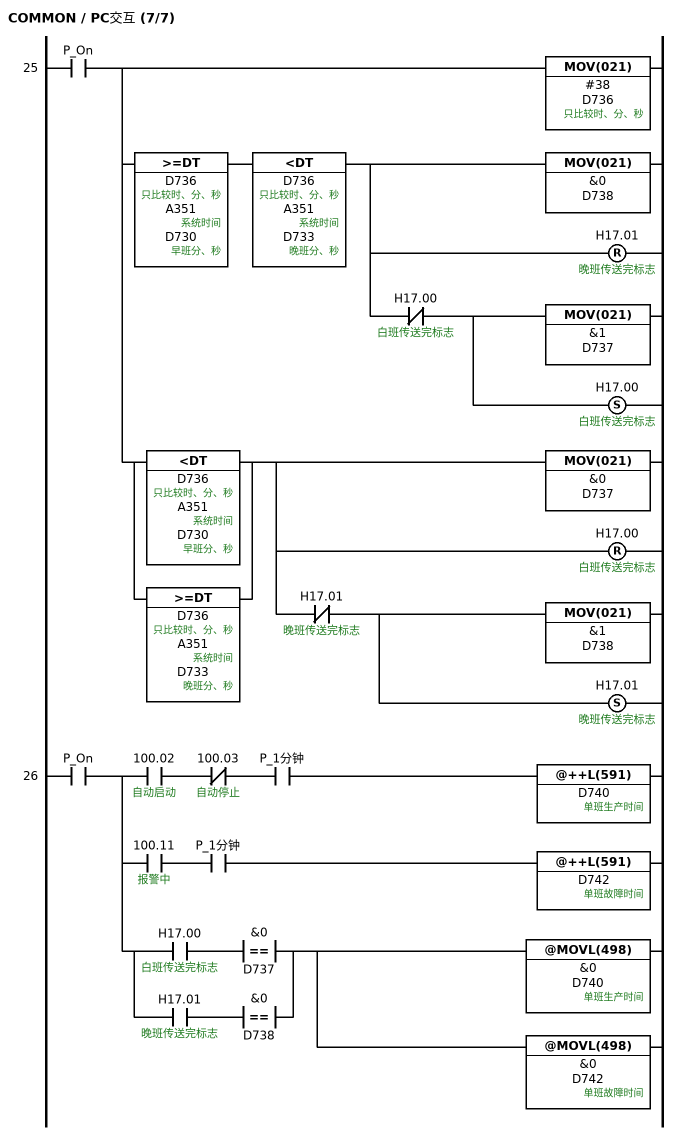
; rung 25
LD P_On
OUT TR0
MOV(021) #38 D736  ; 只比较时、分、秒
AND>=DT(346) D736 A351 D730  ; 只比较时、分、秒, 系统时间, 早班分、秒
AND<DT(343) D736 A351 D733  ; 只比较时、分、秒, 系统时间, 晚班分、秒
MOV(021) &0 D738
RSET H17.01  ; 晚班传送完标志
ANDNOT H17.00  ; 白班传送完标志
MOV(021) &1 D737
SET H17.00  ; 白班传送完标志
LD TR0
LD<DT(343) D736 A351 D730  ; 只比较时、分、秒, 系统时间, 早班分、秒
OR>=DT(346) D736 A351 D733  ; 只比较时、分、秒, 系统时间, 晚班分、秒
ANDLD
MOV(021) &0 D737
RSET H17.00  ; 白班传送完标志
ANDNOT H17.01  ; 晚班传送完标志
MOV(021) &1 D738
SET H17.01  ; 晚班传送完标志
; rung 26
LD P_On
OUT TR0
AND 100.02  ; 自动启动
ANDNOT 100.03  ; 自动停止
AND P_1分钟
@++L(591) D740  ; 单班生产时间
LD TR0
AND 100.11  ; 报警中
AND P_1分钟
@++L(591) D742  ; 单班故障时间
LD TR0
LD H17.00  ; 白班传送完标志
AND=(300) &0 D737
LD H17.01  ; 晚班传送完标志
AND=(300) &0 D738
ORLD
ANDLD
@MOVL(498) &0 D740  ; 单班生产时间
@MOVL(498) &0 D742  ; 单班故障时间

### Section 安东系统

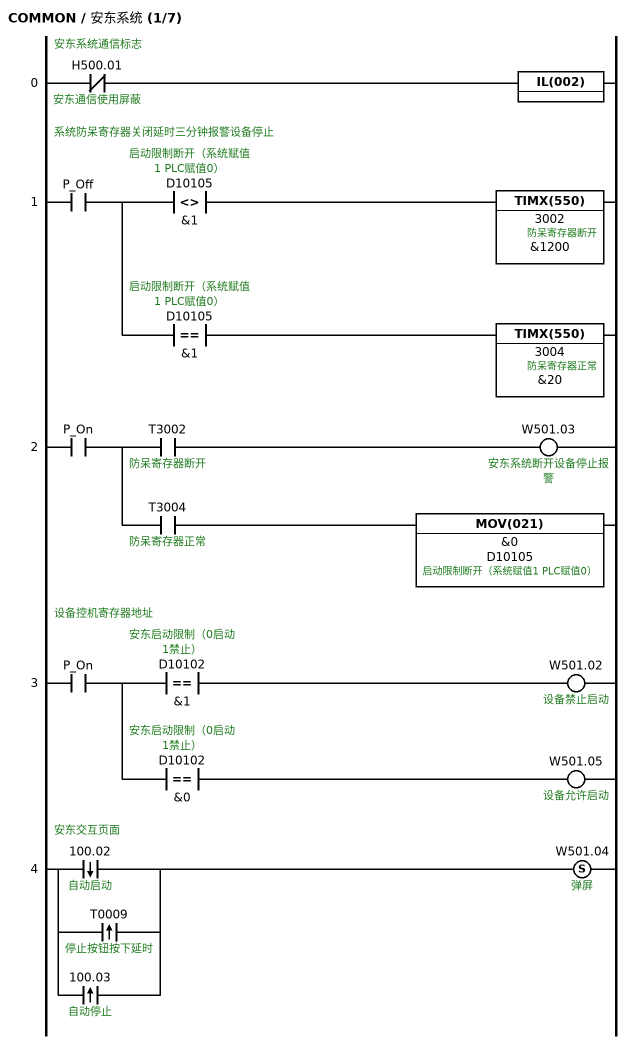
; rung 0: 安东系统通信标志
LDNOT H500.01  ; 安东通信使用屏蔽
IL(002)
; rung 1: 系统防呆寄存器关闭延时三分钟报警设备停止
LD P_Off
OUT TR0
AND<>(305) D10105 &1  ; 启动限制断开（系统赋值1 PLC赋值0）
TIMX(550) 3002 &1200  ; 防呆寄存器断开
LD TR0
AND=(300) D10105 &1  ; 启动限制断开（系统赋值1 PLC赋值0）
TIMX(550) 3004 &20  ; 防呆寄存器正常
; rung 2
LD P_On
OUT TR0
AND T3002  ; 防呆寄存器断开
OUT W501.03  ; 安东系统断开设备停止报警
LD TR0
AND T3004  ; 防呆寄存器正常
MOV(021) &0 D10105  ; 启动限制断开（系统赋值1 PLC赋值0）
; rung 3: 设备控机寄存器地址
LD P_On
OUT TR0
AND=(300) D10102 &1  ; 安东启动限制（0启动 1禁止）
OUT W501.02  ; 设备禁止启动
LD TR0
AND=(300) D10102 &0  ; 安东启动限制（0启动 1禁止）
OUT W501.05  ; 设备允许启动
; rung 4: 安东交互页面
%LD 100.02  ; 自动启动
@OR T0009  ; 停止按钮按下延时
@OR 100.03  ; 自动停止
SET W501.04  ; 弹屏

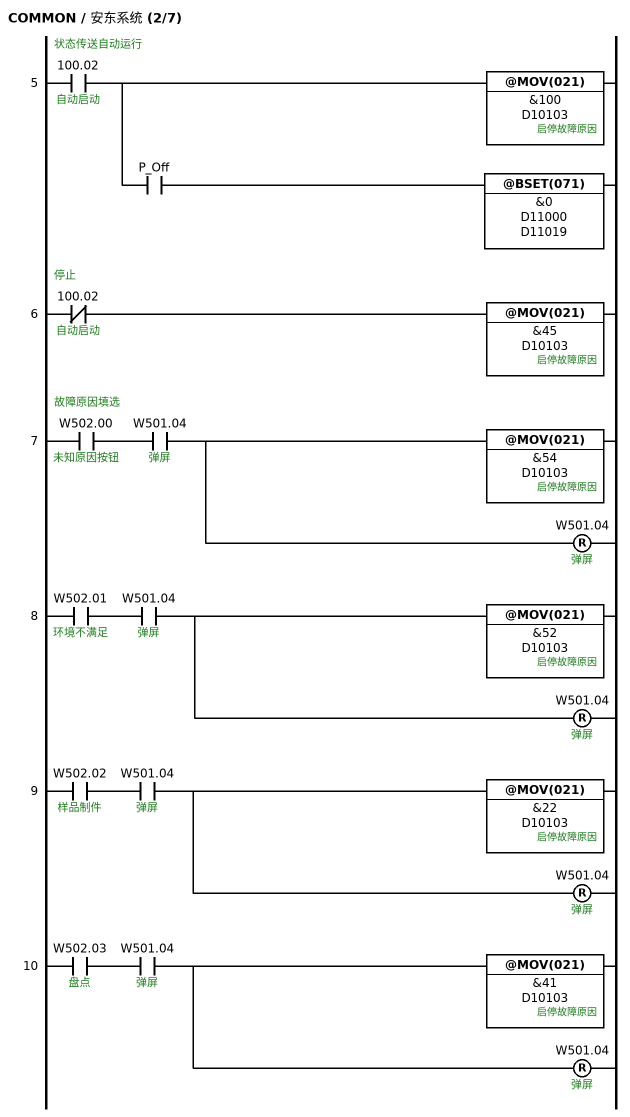
; rung 5: 状态传送自动运行
LD 100.02  ; 自动启动
@MOV(021) &100 D10103  ; 启停故障原因
AND P_Off
@BSET(071) &0 D11000 D11019
; rung 6: 停止
LDNOT 100.02  ; 自动启动
@MOV(021) &45 D10103  ; 启停故障原因
; rung 7: 故障原因填选
LD W502.00  ; 未知原因按钮
AND W501.04  ; 弹屏
@MOV(021) &54 D10103  ; 启停故障原因
RSET W501.04  ; 弹屏
; rung 8
LD W502.01  ; 环境不满足
AND W501.04  ; 弹屏
@MOV(021) &52 D10103  ; 启停故障原因
RSET W501.04  ; 弹屏
; rung 9
LD W502.02  ; 样品制件
AND W501.04  ; 弹屏
@MOV(021) &22 D10103  ; 启停故障原因
RSET W501.04  ; 弹屏
; rung 10
LD W502.03  ; 盘点
AND W501.04  ; 弹屏
@MOV(021) &41 D10103  ; 启停故障原因
RSET W501.04  ; 弹屏

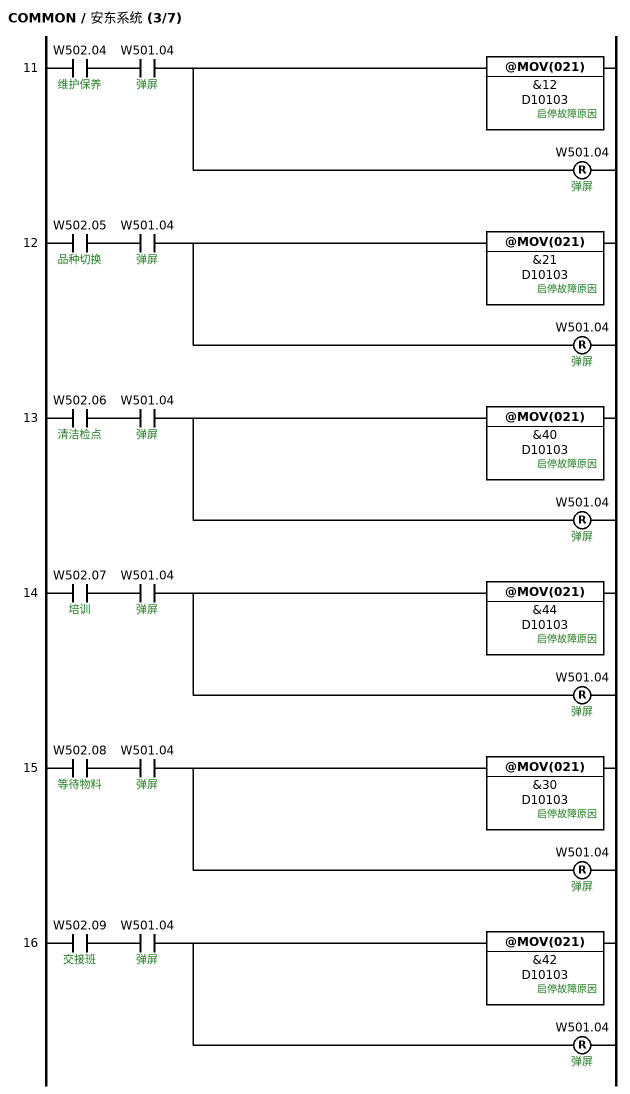
; rung 11
LD W502.04  ; 维护保养
AND W501.04  ; 弹屏
@MOV(021) &12 D10103  ; 启停故障原因
RSET W501.04  ; 弹屏
; rung 12
LD W502.05  ; 品种切换
AND W501.04  ; 弹屏
@MOV(021) &21 D10103  ; 启停故障原因
RSET W501.04  ; 弹屏
; rung 13
LD W502.06  ; 清洁检点
AND W501.04  ; 弹屏
@MOV(021) &40 D10103  ; 启停故障原因
RSET W501.04  ; 弹屏
; rung 14
LD W502.07  ; 培训
AND W501.04  ; 弹屏
@MOV(021) &44 D10103  ; 启停故障原因
RSET W501.04  ; 弹屏
; rung 15
LD W502.08  ; 等待物料
AND W501.04  ; 弹屏
@MOV(021) &30 D10103  ; 启停故障原因
RSET W501.04  ; 弹屏
; rung 16
LD W502.09  ; 交接班
AND W501.04  ; 弹屏
@MOV(021) &42 D10103  ; 启停故障原因
RSET W501.04  ; 弹屏

